(* CODESYS project TcDynStringKit.library
   Company: FisoThemes
   DefaultNamespace: TcDynStringKit
   Version: 1.0.1.1
   Placeholder: TwinCAT Dynamic String Kit
   Author: Goodwill Mzumala
   Description: A library that provides tools for working with dynamic strings in TwinCAT.
   Title: TwinCAT Dynamic String Kit

Project tree, tasks and I/O mapping:
  libraries: Tc2_Standard, * (Beckhoff Automation GmbH); Tc2_System, * (Beckhoff Automation GmbH); Tc2_Utilities, * (Beckhoff Automation GmbH); Tc3_Module, * (Beckhoff Automation GmbH)
  DUTs/
    Alias/
      data type T_Char
      data type T_LongString
      data type T_QueryInterface
      data type T_ShortString
      data type T_Size
      data type T_WhitespaceLocation
    Enums/
      data type E_WhitespaceLocation
    Structs/
    Unions/
  ITFs/
    Adapters/
      interface I_ReadOnlyLineBuilderAdapter
      interface I_ReadOnlyStringBuilderAdapter: Capacity, CopySubstringTo, CopyTo, GetBuffer, GetCapacity, GetChar, GetLength, GetString, GetSubstring, Length, Search, SearchAny, Split
      interface I_ReadOnlyWordBuilderAdapter
    Builders/
      interface I_LineBuilder
      interface I_StringBuilder: Append, AppendAny, AppendBuffer, AppendLine, BTrim, Capacity, Clear, CopySubstringTo, CopyTo, GetBuffer, GetCapacity, GetChar, GetLength, GetString, GetSubstring, Insert, InsertAny, InsertBuffer, Join, Length, LTrim, Remove, Replace, ReplaceAny, Reverse, RTrim, Search, SearchAny, Split, StrinkToFit, ToLowercase, ToUppercase
      interface I_WordBuilder
    Enumerators/
      interface I_Disposable: Dispose
      interface I_Enumerable: GetEnumerator
      interface I_Enumerator: Current, GetCurrent, Next, Reset
  PARAMs/
    GVLs/
      global variables Param_Configurations
  POUs/
    Examples/
      program P_AdapterExample [ST]
      program P_EnumeratorExample [ST]
      program P_StringBuilderExample [ST]
    Function Blocks/
      _Internal/
        function block FB_Free [ST]: FB_exit, FB_init
      Adapters/
        function block FB_ReadOnlyStringBuilderAdapter [ST]: Capacity, CopySubstringTo, CopyTo, GetBuffer, GetCapacity, GetChar, GetEnumerator, GetLength, GetString, GetSubstring, Length, Search, SearchAny, Split
      Builders/
        function block FB_StringBuilder [ST]: Free, Is_Space, Malloc, Reserve, Append, AppendAny, AppendBuffer, AppendLine, BTrim, Capacity, Clear, CopySubstringTo, CopyTo, GetBuffer, GetCapacity, GetChar, GetEnumerator, GetLength, GetString, GetSubstring, Insert, InsertAny, InsertBuffer, Join, Length, LTrim, Remove, Replace, ReplaceAny, Reverse, RTrim, Search, SearchAny, Split, StrinkToFit, ToLowercase, ToUppercase
      Enumerators/
        function block FB_AbstractStringEnumerator [ST]: Current, Dispose, GetCurrent, Next, Reset
        function block FB_StringBuilderEnumerator [ST]: Current, Current_Buffer, FB_init, GetCurrent, Next
    Functions/
      function F_AnyStringLength [ST]
      function F_AnyToString [ST]
      function F_ByteToChar [ST]
      function F_CharToByte [ST]
      function F_IsAnyToStringCompatable [ST]
      function F_IsBool [ST]
      function F_IsDigit [ST]
      function F_IsLTime [ST]
      function F_IsNumber [ST]
      function F_IsSignedInteger [ST]
      function F_IsSpace [ST]
      function F_IsTime [ST]
      function F_IsUnsignedInteger [ST]
      function F_MallocStr [ST]
      function F_MemCpy [ST]
      function F_MemMove [ST]
      function F_StringBuilder [ST]
      function F_StrLCat [ST]
      function F_StrLCpy [ST]
      function F_StrLen [ST]
      function F_StrNCmp [ST]
      function F_StrStr [ST]
      function F_StrToAny [ST]
      function F_ToLower [ST]
      function F_ToUpper [ST]
      function F_TrimWhiteSpace [ST]
    program MAIN [ST]
  Project Information/
    function F_GetCompany [ST]
    function F_GetTitle [ST]
    function F_GetVersion [ST]
  Version/
    global variables Global_Version
  VISUs/
*)

// DUTs/Alias/T_Char
TYPE T_Char : STRING(1); END_TYPE

// DUTs/Alias/T_LongString
TYPE T_LongString : STRING(Param_Configurations.LongStringSize); END_TYPE

// DUTs/Alias/T_QueryInterface
TYPE T_QueryInterface : __SYSTEM.IQueryInterface; END_TYPE

// DUTs/Alias/T_ShortString
TYPE T_ShortString : STRING(Param_Configurations.ShortStringSize); END_TYPE

// DUTs/Alias/T_Size
TYPE T_Size : DINT; END_TYPE

// DUTs/Alias/T_WhitespaceLocation
TYPE T_WhitespaceLocation : E_WhitespaceLocation; END_TYPE

// DUTs/Enums/E_WhitespaceLocation
{attribute 'qualified_only'}
{attribute 'to_string'}
TYPE E_WhitespaceLocation :
(
	Both := 0,
	Start,
	End
);
END_TYPE

// PARAMs/GVLs/Param_Configurations
{attribute 'qualified_only'}
VAR_GLOBAL CONSTANT
	ShortStringSize : UXINT := 80;
	LongStringSize : UXINT := 255;
END_VAR

// Version/Global_Version
{attribute 'TcGenerated'}
{attribute 'no-analysis'}
{attribute 'linkalways'}
// This function has been automatically generated from the project information.
VAR_GLOBAL CONSTANT
	{attribute 'const_non_replaced'}
	stLibVersion_TwinCAT_Dynamic_String_Kit : ST_LibVersion := (iMajor := 1, iMinor := 0, iBuild := 1, iRevision := 1, nFlags := 0, sVersion := '1.0.1.1');
END_VAR

// ITFs/Adapters/I_ReadOnlyLineBuilderAdapter
INTERFACE I_ReadOnlyLineBuilderAdapter EXTENDS T_QueryInterface

END_INTERFACE

// ITFs/Adapters/I_ReadOnlyStringBuilderAdapter
INTERFACE I_ReadOnlyStringBuilderAdapter EXTENDS T_QueryInterface

// Number of bytes allocated in memory for the string builder's contents.
PROPERTY Capacity : T_Size
GET
END_GET
END_PROPERTY

// Copies a subset of characters in the string builder from specified position at specified length to a string
METHOD CopySubstringTo : I_ReadOnlyStringBuilderAdapter
VAR_INPUT
	Position, Length : T_Size;
	Value : ANY;
END_VAR
END_METHOD

// Copies contents of string builder to given string of any size
METHOD CopyTo : I_ReadOnlyStringBuilderAdapter
VAR_INPUT
	Value : ANY;
END_VAR
END_METHOD

// !!!UNSAFE!!! DON'T FORGET TO RELEASE/DELETE FROM	MEMORY WHEN DONE!
// | Get a copy of the internal string buffer at the size of the string length + 1.
METHOD GetBuffer : I_ReadOnlyStringBuilderAdapter
VAR_IN_OUT
	pBuffer : POINTER TO BYTE;
END_VAR
END_METHOD

// Retrieves the number of bytes allocated in memory for the string builder's contents.
METHOD GetCapacity : I_ReadOnlyStringBuilderAdapter
VAR_OUTPUT
	Capacity : T_Size;
END_VAR
END_METHOD

// Gets character at specified position in the string builder
METHOD GetChar : T_Char
VAR_INPUT
	Position : T_Size;
END_VAR
END_METHOD

// Retrieves the current size of string builder contents
METHOD GetLength : I_ReadOnlyStringBuilderAdapter
VAR_OUTPUT
	Length : T_Size;
END_VAR
END_METHOD

// Converts contents of string builder to string and returns them
METHOD GetString : T_LongString
VAR_INPUT
END_VAR
END_METHOD

// Get a subset of characters in the string builder from specified position at specified length and returns them as a string
METHOD GetSubstring : T_LongString
VAR_INPUT
	Position, Length : T_Size;
END_VAR
END_METHOD

// Current size of string builder contents
PROPERTY Length : T_Size
GET
END_GET
END_PROPERTY

// Finds the position of the first instance of a given string in the content's of the string builder from a starting position
METHOD Search : I_ReadOnlyStringBuilderAdapter
VAR_INPUT
	sValue : T_LongString;
	Start_Position : T_Size;
END_VAR
VAR_OUTPUT
	Position : T_Size;
END_VAR
END_METHOD

// Finds the position of the first instance of a given value in the content's of the string builder from a starting position
METHOD SearchAny : I_ReadOnlyStringBuilderAdapter
VAR_INPUT
	Value : ANY;
	Start_Position : T_Size;
END_VAR
VAR_OUTPUT
	Position : T_Size := -1;
END_VAR
END_METHOD

// Appends selected characters from the current string builder to the selected string builder
METHOD Split : I_ReadOnlyStringBuilderAdapter
VAR_INPUT
	Position, Length : T_Size;
	ipStringBuilder : I_StringBuilder;
END_VAR
END_METHOD

END_INTERFACE

// ITFs/Builders/I_StringBuilder
INTERFACE I_StringBuilder EXTENDS T_QueryInterface

// Appends the given string to the end of the string builder's contents.
METHOD Append : I_StringBuilder
VAR_INPUT
	sValue : T_LongString;
END_VAR
END_METHOD

// Appends the given value to the end of the string builder's contents.
METHOD AppendAny : I_StringBuilder
VAR_INPUT
	Value : ANY;
END_VAR
END_METHOD

// !!!UNSAFE!!! THIS WILL APPEND UP TO THE NULL CHARACTER. IF NO NULL EXISTS, THIS WILL RUN FOREVER!
// | Append raw values directly to the internal string buffer. This is meant for appending dynamic strings to the string builder.
METHOD AppendBuffer : I_StringBuilder
VAR_INPUT
	pBuffer : POINTER TO BYTE;
END_VAR
END_METHOD

// Appends a new line (\r\n or $r$n) to string builder's contents.
METHOD AppendLine : I_StringBuilder
END_METHOD

// Removes all ASCII white space (spaces, tabs, carriage returns, and linefeeds) from the beginning and end of string in the string builder
METHOD BTrim : I_StringBuilder
END_METHOD

// Number of bytes allocated in memory for the string builder's contents.
PROPERTY Capacity : T_Size
GET
END_GET
END_PROPERTY

// Empties the string builder's contents, resetting its length to zero.
METHOD Clear : I_StringBuilder
END_METHOD

// Copies a subset of characters in the string builder from specified position at specified length to a string
METHOD CopySubstringTo : I_StringBuilder
VAR_INPUT
	Position, Length : T_Size;
	Value : ANY;
END_VAR
END_METHOD

// Copies contents of string builder to given string of any size
METHOD CopyTo : I_StringBuilder
VAR_INPUT
	Value : ANY;
END_VAR
END_METHOD

// !!!UNSAFE!!! DON'T FORGET TO RELEASE/DELETE FROM	MEMORY WHEN DONE!
// | Get a copy of the internal string buffer at the size of the string length + 1.
METHOD GetBuffer : I_StringBuilder
VAR_IN_OUT
	pBuffer : POINTER TO BYTE;
END_VAR
END_METHOD

// Retrieves the number of bytes allocated in memory for the string builder's contents.
METHOD GetCapacity : I_StringBuilder
VAR_OUTPUT
	Capacity : T_Size;
END_VAR
END_METHOD

// Gets character at specified position in the string builder
METHOD GetChar : T_Char
VAR_INPUT
	Position : T_Size;
END_VAR
END_METHOD

// Retrieves the current size of string builder contents
METHOD GetLength : I_StringBuilder
VAR_OUTPUT
	Length : T_Size;
END_VAR
END_METHOD

// Converts contents of string builder to string and returns them
METHOD GetString : T_LongString
VAR_INPUT
END_VAR
END_METHOD

// Get a subset of characters in the string builder from specified position at specified length and returns them as a string
METHOD GetSubstring : T_LongString
VAR_INPUT
	Position, Length : T_Size;
END_VAR
END_METHOD

// Inserts the given string at the specified position.
METHOD Insert : I_StringBuilder
VAR_INPUT
	Position : T_Size;
	sValue : T_LongString;
END_VAR
END_METHOD

// Inserts the given value at the specified position.
METHOD InsertAny : I_StringBuilder
VAR_INPUT
	Position : T_Size;
	Value : ANY;
END_VAR
END_METHOD

// !!!UNSAFE!!! THIS WILL INSERT UP TO THE NULL CHARACTER. IF NO NULL EXISTS, THIS WILL RUN FOREVER!
// | Inserts raw values directly to the internal string buffer at the specified position. This is meant for inserting dynamic strings to the string builder.
METHOD InsertBuffer : I_StringBuilder
VAR_INPUT
	Position : T_Size;
	pBuffer : POINTER TO BYTE;
END_VAR
END_METHOD

// Joins/Merges the string contents of the current string builder with that on the specified string builder at the specified position
METHOD Join : I_StringBuilder
VAR_INPUT
	Position : T_Size;
	ipString_Builder : I_StringBuilder;
END_VAR
END_METHOD

// Current size of string builder contents
PROPERTY Length : T_Size
GET
END_GET
END_PROPERTY

// Removes all ASCII white space (spaces, tabs, carriage returns, and linefeeds) from the beginning of string in the string builder
METHOD LTrim : I_StringBuilder
VAR_INPUT
END_VAR
END_METHOD

// Removes the characters in the string builder from specified position at specified length.
METHOD Remove : I_StringBuilder
VAR_INPUT
	Position, Length : T_Size;
END_VAR
END_METHOD

// Replaces the instance of the old string in the string builder with the new string.
// If bReplace_All = TRUE, all instances of the old string are placed, else only the first instance.
METHOD Replace : I_StringBuilder
VAR_INPUT
	sOld_Value,
	sNew_Value : T_LongString;
	bReplace_All : BOOL;
END_VAR
END_METHOD

// Replaces the instance of the old value in the string builder with the new value.
// If bReplace_All = TRUE, all instances of the old value are placed, else only the first instance.
METHOD ReplaceAny : I_StringBuilder
VAR_INPUT
	Old_Value : ANY;
	New_Value : ANY;
	bReplace_All : BOOL;
END_VAR
END_METHOD

// Reverses the string contents in the string builder
METHOD Reverse : I_StringBuilder
VAR_INPUT
END_VAR
END_METHOD

// Removes all ASCII white space (spaces, tabs, carriage returns, and linefeeds) from the end of string in the string builder
METHOD RTrim : I_StringBuilder
VAR_INPUT
END_VAR
END_METHOD

// Finds the position of the first instance of a given string in the content's of the string builder from a starting position
METHOD Search : I_StringBuilder
VAR_INPUT
	sValue : T_LongString;
	Start_Position : T_Size;
END_VAR
VAR_OUTPUT
	Position : T_Size;
END_VAR
END_METHOD

// Finds the position of the first instance of a given value in the content's of the string builder from a starting position
METHOD SearchAny : I_StringBuilder
VAR_INPUT
	Value : ANY;
	Start_Position : T_Size;
END_VAR
VAR_OUTPUT
	Position : T_Size := -1;
END_VAR
END_METHOD

// Appends selected characters from the current string builder to the selected string builder
METHOD Split : I_StringBuilder
VAR_INPUT
	Position, Length : T_Size;
	ipStringBuilder : I_StringBuilder;
END_VAR
END_METHOD

// Reduces the capacity of the string builder to match the size of its contents, potentially reducing memory usage.
METHOD StrinkToFit : I_StringBuilder
END_METHOD

// Converts all alphabetic characters in string builder to lowercase characters
METHOD ToLowercase : I_StringBuilder
VAR_INPUT
END_VAR
END_METHOD

// Converts all alphabetic characters in string builder to uppercase characters
METHOD ToUppercase : I_StringBuilder
VAR_INPUT
END_VAR
END_METHOD

END_INTERFACE

// ITFs/Adapters/I_ReadOnlyWordBuilderAdapter
INTERFACE I_ReadOnlyWordBuilderAdapter EXTENDS T_QueryInterface

END_INTERFACE

// ITFs/Builders/I_LineBuilder
INTERFACE I_LineBuilder EXTENDS T_QueryInterface

END_INTERFACE

// ITFs/Builders/I_WordBuilder
INTERFACE I_WordBuilder EXTENDS T_QueryInterface

END_INTERFACE

// ITFs/Enumerators/I_Disposable
INTERFACE I_Disposable EXTENDS T_QueryInterface

// Disposes or release resources for specified task
METHOD Dispose
VAR_INPUT
END_VAR
END_METHOD

END_INTERFACE

// ITFs/Enumerators/I_Enumerable
INTERFACE I_Enumerable EXTENDS T_QueryInterface

METHOD GetEnumerator : I_Enumerator
VAR_INPUT
END_VAR
END_METHOD

END_INTERFACE

// ITFs/Enumerators/I_Enumerator
INTERFACE I_Enumerator EXTENDS I_Disposable

(* Gets current string representation of element*)
PROPERTY Current : T_LongString
GET
END_GET
END_PROPERTY

// Gets current element. Returns TRUE if retrieval and converstion was successful.
METHOD GetCurrent : BOOL
VAR_INPUT
	sValue : REFERENCE TO STRING;
END_VAR
END_METHOD

// Advances enumerator to the next element. On first call or after reset it generates new element data to enumerate over.
METHOD Next : BOOL
VAR_INPUT
END_VAR
END_METHOD

// Sets enumerator to it's intial position. Disposes data pertaining to it's old elements.
METHOD Reset
VAR_INPUT
END_VAR
END_METHOD

END_INTERFACE

// POUs/Examples/P_AdapterExample
PROGRAM INTERNAL P_AdapterExample
VAR
	bStart				: BOOL;
	sValue 				: STRING(255);
	nPos				: T_Size;
	tTime 				: TIME :=  TIME();
	tTime2				: TIME;
	fbStringBuilder 	: FB_StringBuilder;
	fbReadOnlySB 		: FB_ReadOnlyStringBuilderAdapter;
	ipReadOnlySB 		: I_ReadOnlyStringBuilderAdapter;
END_VAR

fbReadOnlySB(ipStringBuilder := fbStringBuilder);
ipReadOnlySB := fbReadOnlySB;

IF bStart THEN
	bStart := FALSE;
	fbStringBuilder
		.Clear()
		.Append('   I love cats.')
		.Append('The time is: ').AppendAny(tTime).Append('.')
		.Append('   ')
		.BTrim();
	END_IF

sValue := ipReadOnlySB
			.Search('T#', 0, Position => nPos)
			.CopySubstringTo(nPos, tc2_Standard.LEN(TO_STRING(tTime)), tTime2)
			.GetString();

END_PROGRAM

// POUs/Function Blocks/Builders/FB_StringBuilder
{attribute 'no_assign'}
{attribute 'enable_dynamic_creation'}
{attribute 'no_explicit_call' := 'do not call this POU directly'}
FUNCTION_BLOCK FB_StringBuilder IMPLEMENTS I_StringBuilder, I_Enumerable
VAR CONSTANT
	Default_Capacity : T_Size := 256;
END_VAR
VAR
	{attribute 'hide'} 
	_Capacity : T_Size := THIS^.Default_Capacity;
	{attribute 'hide'} 
	_Length : T_Size := 0;
	_pBuffer : POINTER TO STRING := THIS^.Malloc(THIS^.Capacity);
END_VAR
VAR CONSTANT
	{attribute 'hide'} 
	_fbFree : FB_Free(THIS^._pBuffer) := ();
END_VAR

// Dealloocates String from memory
METHOD PROTECTED Free
VAR_INPUT
END_VAR
IF THIS^._pBuffer <> 0 THEN __DELETE(THIS^._pBuffer); END_IF
THIS^.Capacity := 0;
END_METHOD

METHOD PROTECTED Is_Space : BOOL
VAR_INPUT
	nChar : BYTE;
END_VAR
Is_Space := (nChar = 32) OR_ELSE (nChar = 9) OR_ELSE (nChar = 10) OR_ELSE (nChar = 13) OR_ELSE (nChar = 12) OR_ELSE (nChar = 11);
END_METHOD

// Allocates memory on the heap for a string of defined size
METHOD PROTECTED Malloc : POINTER TO STRING
VAR_INPUT
	Size : T_Size;
END_VAR
Malloc := __NEW(BYTE, TO_UDINT(Size));
END_METHOD

METHOD PROTECTED Reserve
VAR_INPUT
	Capacity : T_Size;
END_VAR
VAR
	pTemp : POINTER TO STRING;
END_VAR
IF Capacity <= THIS^.Capacity THEN RETURN; END_IF
pTemp := THIS^.Malloc(Capacity);
F_StrLCpy(pTemp, THIS^._pBuffer, Capacity);
THIS^.Free();
THIS^._pBuffer := pTemp;
THIS^.Capacity := Capacity;
END_METHOD

// Appends the given string to the end of the string builder's contents.
METHOD Append : I_StringBuilder
VAR_INPUT
	sValue : T_LongString;
END_VAR
Append := THIS^.AppendAny(sValue);
END_METHOD

// Appends the given value to the end of the string builder's contents.
METHOD AppendAny : I_StringBuilder
VAR_INPUT
	Value : ANY;
END_VAR
VAR
	bMalloced : BOOL := TRUE;
	Str_Len : T_Size;
	pValue : POINTER TO STRING;
END_VAR
AppendAny := THIS^;
CASE Value.TypeClass OF
	__SYSTEM.TYPE_CLASS.TYPE_STRING: 
		Str_Len := F_StrLen(Value.pValue);
		pValue := Value.pValue;
		bMalloced := FALSE;
		
	__SYSTEM.TYPE_CLASS.TYPE_WSTRING:
		Str_Len := TO_DINT(Tc2_Utilities.WLEN2(Value.pValue));
		pValue := THIS^.Malloc(Str_Len);
		Tc2_Utilities.WSTRING_TO_STRING2(pValue, Value.pValue, TO_UDINT(Str_Len));
		
	__SYSTEM.TYPE_CLASS.TYPE_BOOL,
	__SYSTEM.TYPE_CLASS.TYPE_BYTE,
	__SYSTEM.TYPE_CLASS.TYPE_WORD,
	__SYSTEM.TYPE_CLASS.TYPE_DWORD,
	__SYSTEM.TYPE_CLASS.TYPE_LWORD,
	__SYSTEM.TYPE_CLASS.TYPE_SINT,
	__SYSTEM.TYPE_CLASS.TYPE_INT,
	__SYSTEM.TYPE_CLASS.TYPE_DINT,
	__SYSTEM.TYPE_CLASS.TYPE_LINT,
	__SYSTEM.TYPE_CLASS.TYPE_USINT,
	__SYSTEM.TYPE_CLASS.TYPE_UINT,
	__SYSTEM.TYPE_CLASS.TYPE_UDINT,
	__SYSTEM.TYPE_CLASS.TYPE_ULINT,
	__SYSTEM.TYPE_CLASS.TYPE_REAL,
	__SYSTEM.TYPE_CLASS.TYPE_LREAL,
	__SYSTEM.TYPE_CLASS.TYPE_TIME,
	__SYSTEM.TYPE_CLASS.TYPE_LTIME,
	__SYSTEM.TYPE_CLASS.TYPE_DATE,
	__SYSTEM.TYPE_CLASS.TYPE_DATEANDTIME,
	__SYSTEM.TYPE_CLASS.TYPE_TIMEOFDAY,
	__SYSTEM.TYPE_CLASS.TYPE_POINTER:
		pValue := THIS^.Malloc(SIZEOF(T_LongString));
		pValue^ := F_AnyToString(Value);
		Str_Len := F_StrLen(pValue);
ELSE
	RETURN;
END_CASE

IF (THIS^.Length + Str_Len) >= THIS^.Capacity THEN
	THIS^.Reserve((THIS^.Length + Str_Len + 1)*2);
	END_IF

THIS^.Length := THIS^.Length + Str_Len;
F_StrLCat(THIS^._pBuffer, pValue, THIS^.Length + 1);

IF bMalloced THEN __DELETE(pValue); END_IF
END_METHOD

// !!!UNSAFE!!! THIS WILL APPEND UP TO THE NULL CHARACTER. IF NO NULL EXISTS, THIS WILL RUN FOREVER!
// | Append raw values directly to the internal string buffer. This is meant for appending dynamic strings to the string builder.
METHOD AppendBuffer : I_StringBuilder
VAR_INPUT
	pBuffer : POINTER TO BYTE;
END_VAR
VAR
	Str_Len : T_Size;
END_VAR
AppendBuffer := THIS^;
IF pBuffer = 0 THEN RETURN; END_IF
Str_Len := F_StrLen(pBuffer);

IF (THIS^.Length + Str_Len) >= THIS^.Capacity THEN
	THIS^.Reserve((THIS^.Length + Str_Len + 1)*2);
	END_IF
	
THIS^.Length := THIS^.Length + Str_Len;
F_StrLCat(THIS^._pBuffer, pBuffer, THIS^.Length + 1);
END_METHOD

// Appends a new line (\r\n or $r$n) to string builder's contents.
METHOD AppendLine : I_StringBuilder
AppendLine := THIS^;
THIS^.Append('$r$n');
END_METHOD

// Removes all ASCII white space (spaces, tabs, carriage returns, and linefeeds) from the beginning and end of string in the string builder
METHOD BTrim : I_StringBuilder
VAR
	Start, End, Length : T_Size := 0;
END_VAR
BTrim := THIS^;
IF THIS^.Length = 0 THEN RETURN; END_IF
End := THIS^.Length - 1;

WHILE ((Start <= End) AND THIS^.Is_Space(THIS^._pBuffer^[Start])) DO Start := Start  + 1; END_WHILE
WHILE ((End >= Start) AND THIS^.Is_Space(THIS^._pBuffer^[End])) DO End := End  - 1; END_WHILE

Length := end - start + 1;
F_MemMove(THIS^._pBuffer, ADR(THIS^._pBuffer^[Start]), Length);
THIS^.Length := Length;
THIS^._pBuffer^[THIS^.Length] := 0;
END_METHOD

// Number of bytes allocated in memory for the string builder's contents.
PROPERTY Capacity : T_Size
GET
Capacity := THIS^._Capacity;
END_GET
SET
PROTECTED
THIS^._Capacity := Capacity;
END_SET
END_PROPERTY

// Empties the string builder's contents, resetting its length to zero.
METHOD Clear : I_StringBuilder
Clear := THIS^;
THIS^.Free();
THIS^.Capacity := THIS^.Default_Capacity;
THIS^.Length := 0;
THIS^._pBuffer := THIS^.Malloc(THIS^.Capacity);
THIS^._pBuffer^[0] := 0;
END_METHOD

// Copies a subset of characters in the string builder from specified position at specified length to a string
METHOD CopySubstringTo : I_StringBuilder
VAR_INPUT
	Position, Length : T_Size;
	Value : ANY;
END_VAR
VAR
	pTemp : POINTER TO BYTE;
	pwsTemp : POINTER TO WSTRING;
END_VAR
CopySubstringTo := THIS^;
IF Value.pValue = 0 THEN RETURN; END_IF
CASE Value.TypeClass OF
	__SYSTEM.TYPE_CLASS.TYPE_STRING:
		Length := MIN(Length, Value.diSize - 1);
		IF (Position > THIS^.Length) OR_ELSE (Length <= 0) OR_ELSE (THIS^.Length = 0) THEN Value.pValue[0] := 0; RETURN; END_IF
		F_StrLCpy(Value.pValue, ADR(THIS^._pBuffer^[Position]), Length + 1);
		
	__SYSTEM.TYPE_CLASS.TYPE_WSTRING:
		Length := MIN(Length, (Value.diSize/2) - 1 );
		IF (Position > THIS^.Length) OR_ELSE (Length = 0) OR_ELSE (THIS^.Length = 0) THEN pwsTemp := Value.pValue; pwsTemp^ := ""; RETURN; END_IF
		pTemp := THIS^.Malloc(Length + 1);
		F_StrLCpy(pTemp, ADR(THIS^._pBuffer^[Position]), Length + 1);
		Tc2_Utilities.STRING_TO_WSTRING2(Value.pValue, pTemp, TO_UDINT((Length*2)+1));
		__DELETE(pTemp);
ELSE
	F_StrToAny(Value, THIS^.GetSubstring(Position, Length));
END_CASE
END_METHOD

// Copies contents of string builder to given string of any size
METHOD CopyTo : I_StringBuilder
VAR_INPUT
	Value : ANY;
END_VAR
CopyTo := THIS^;
IF THIS^._pBuffer = 0 THEN Value.pValue[0] := 0; RETURN; END_IF 
CASE Value.TypeClass OF
	__SYSTEM.TYPE_CLASS.TYPE_STRING:
		F_StrLCpy(Value.pValue, THIS^._pBuffer, Value.diSize);
	__SYSTEM.TYPE_CLASS.TYPE_WSTRING:
		Tc2_Utilities.STRING_TO_WSTRING2(Value.pValue, THIS^._pBuffer, TO_UDINT(Value.diSize));
ELSE
	F_StrToAny(Value, THIS^.GetString());
END_CASE
END_METHOD

// !!!UNSAFE!!! DON'T FORGET TO RELEASE/DELETE FROM	MEMORY WHEN DONE!
// | Get a copy of the internal string buffer at the size of the string length + 1.
METHOD GetBuffer : I_StringBuilder
VAR_IN_OUT
	pBuffer : POINTER TO BYTE;
END_VAR
GetBuffer := THIS^;
pBuffer := THIS^.Malloc(THIS^.Length + 1);
F_StrLCpy(pBuffer, THIS^._pBuffer, THIS^.Length + 1);
END_METHOD

// Retrieves the number of bytes allocated in memory for the string builder's contents.
METHOD GetCapacity : I_StringBuilder
VAR_OUTPUT
	Capacity : T_Size;
END_VAR
GetCapacity := THIS^;
Capacity := THIS^.Capacity;
END_METHOD

// Gets character at specified position in the string builder
METHOD GetChar : T_Char
VAR_INPUT
	Position : T_Size;
END_VAR
IF Position < 0 THEN RETURN; END_IF
IF Position > THIS^.Length THEN RETURN; END_IF
GetChar[0] := THIS^._pBuffer^[Position];
END_METHOD

METHOD GetEnumerator : I_Enumerator
VAR_INST
	fbEnumerator : FB_StringBuilderEnumerator(THIS^);
END_VAR
GetEnumerator := fbEnumerator;
END_METHOD

// Retrieves the current size of string builder contents
METHOD GetLength : I_StringBuilder
VAR_OUTPUT
	Length : T_Size;
END_VAR
GetLength := THIS^;
Length := THIS^.Length;
END_METHOD

// Converts contents of string builder to string and returns them
METHOD GetString : T_LongString
THIS^.CopyTo(GetString);
END_METHOD

// Get a subset of characters in the string builder from specified position at specified length and returns them as a string
METHOD GetSubstring : T_LongString
VAR_INPUT
	Position, Length : T_Size;
END_VAR
THIS^.CopySubstringTo(Position, Length, GetSubstring);
END_METHOD

// Inserts the given string at the specified position.
METHOD Insert : I_StringBuilder
VAR_INPUT
	Position : T_Size;
	sValue : T_LongString;
END_VAR
Insert := THIS^.InsertAny(Position, sValue);
END_METHOD

// Inserts the given value at the specified position.
METHOD InsertAny : I_StringBuilder
VAR_INPUT
	Position : T_Size;
	Value : ANY;
END_VAR
VAR
	bMalloced : BOOL := TRUE;
	Str_Len : T_Size;
	pValue : POINTER TO STRING;
END_VAR
InsertAny := THIS^;
IF Position < 0 OR Position > THIS^.Length THEN RETURN; END_IF 
CASE Value.TypeClass OF
	__SYSTEM.TYPE_CLASS.TYPE_STRING: 
		Str_Len := F_StrLen(Value.pValue);
		pValue := Value.pValue;
		bMalloced := FALSE;
	
	__SYSTEM.TYPE_CLASS.TYPE_WSTRING:
		Str_Len := TO_DINT(Tc2_Utilities.WLEN2(Value.pValue));
		pValue := THIS^.Malloc(Str_Len);
		Tc2_Utilities.WSTRING_TO_STRING2(pValue, Value.pValue, TO_UDINT(Str_Len));

	__SYSTEM.TYPE_CLASS.TYPE_BOOL,
	__SYSTEM.TYPE_CLASS.TYPE_BYTE,
	__SYSTEM.TYPE_CLASS.TYPE_WORD,
	__SYSTEM.TYPE_CLASS.TYPE_DWORD,
	__SYSTEM.TYPE_CLASS.TYPE_LWORD,
	__SYSTEM.TYPE_CLASS.TYPE_SINT,
	__SYSTEM.TYPE_CLASS.TYPE_INT,
	__SYSTEM.TYPE_CLASS.TYPE_DINT,
	__SYSTEM.TYPE_CLASS.TYPE_LINT,
	__SYSTEM.TYPE_CLASS.TYPE_USINT,
	__SYSTEM.TYPE_CLASS.TYPE_UINT,
	__SYSTEM.TYPE_CLASS.TYPE_UDINT,
	__SYSTEM.TYPE_CLASS.TYPE_ULINT,
	__SYSTEM.TYPE_CLASS.TYPE_REAL,
	__SYSTEM.TYPE_CLASS.TYPE_LREAL,
	__SYSTEM.TYPE_CLASS.TYPE_TIME,
	__SYSTEM.TYPE_CLASS.TYPE_LTIME,
	__SYSTEM.TYPE_CLASS.TYPE_DATE,
	__SYSTEM.TYPE_CLASS.TYPE_DATEANDTIME,
	__SYSTEM.TYPE_CLASS.TYPE_TIMEOFDAY,
	__SYSTEM.TYPE_CLASS.TYPE_POINTER:
		pValue := THIS^.Malloc(SIZEOF(T_LongString));
		pValue^ := F_AnyToString(Value);
		Str_Len := F_StrLen(pValue);
ELSE
	RETURN;
END_CASE

IF (THIS^.Length + Str_Len) >= THIS^.Capacity THEN
	THIS^.Reserve((THIS^.Length + Str_Len + 1)*2);
	END_IF

F_MemMove(THIS^._pBuffer + TO_UDINT(Position) + TO_UDINT(Str_Len), THIS^._pBuffer + TO_UDINT(Position), THIS^.Length - Position + 1);
F_MemCpy(THIS^._pBuffer + TO_UDINT(Position), pValue, Str_Len); 
THIS^.Length := THIS^.Length + Str_Len;

IF bMalloced THEN __DELETE(pValue); END_IF
END_METHOD

// !!!UNSAFE!!! THIS WILL INSERT UP TO THE NULL CHARACTER. IF NO NULL EXISTS, THIS WILL RUN FOREVER!
// | Inserts raw values directly to the internal string buffer at the specified position. This is meant for inserting dynamic strings to the string builder.
METHOD InsertBuffer : I_StringBuilder
VAR_INPUT
	Position : T_Size;
	pBuffer : POINTER TO BYTE;
END_VAR
VAR
	Str_Len : T_Size;
END_VAR
InsertBuffer := THIS^;
IF pBuffer = 0 OR Position < 0 OR Position > THIS^.Length THEN RETURN; END_IF
Str_Len := F_StrLen(pBuffer);

IF (THIS^.Length + Str_Len) >= THIS^.Capacity THEN
	THIS^.Reserve((THIS^.Length + Str_Len + 1)*2);
	END_IF

F_MemMove(THIS^._pBuffer + TO_UDINT(Position) + TO_UDINT(Str_Len), THIS^._pBuffer + TO_UDINT(Position), THIS^.Length - Position + 1);
F_MemCpy(THIS^._pBuffer + TO_UDINT(Position), pBuffer, Str_Len); 
THIS^.Length := THIS^.Length + Str_Len;
END_METHOD

// Joins/Merges the string contents of the current string builder with that on the specified string builder at the specified position
METHOD Join : I_StringBuilder
VAR_INPUT
	Position : T_Size;
	ipString_Builder : I_StringBuilder;
END_VAR
VAR
	pTemp : POINTER TO BYTE;
END_VAR
Join := THIS^;
IF ipString_Builder = 0 THEN RETURN; END_IF
ipString_Builder.GetBuffer(pTemp);
THIS^.InsertBuffer(Position, pTemp);
CASE Tc2_System.F_CheckMemoryArea(pTemp, 1) OF 
	E_TcMemoryArea.Dynamic: __DELETE(pTemp);
END_CASE
END_METHOD

// Current size of string builder contents
PROPERTY Length : T_Size
GET
VAR
	i : UDINT;
END_VAR
Length := THIS^._Length;
END_GET
SET
PROTECTED 
VAR
END_VAR
THIS^._Length := Length;
END_SET
END_PROPERTY

// Removes all ASCII white space (spaces, tabs, carriage returns, and linefeeds) from the beginning of string in the string builder
METHOD LTrim : I_StringBuilder
VAR
	Start, End, Length : T_Size := 0;
END_VAR
LTrim := THIS^;
IF THIS^.Length = 0 THEN RETURN; END_IF
End := THIS^.Length - 1;

WHILE ((Start <= End) AND THIS^.Is_Space(THIS^._pBuffer^[Start])) DO Start := Start + 1; END_WHILE

Length := end - start + 1;
F_MemMove(THIS^._pBuffer, ADR(THIS^._pBuffer^[Start]), Length);
THIS^.Length := Length;
THIS^._pBuffer^[THIS^.Length] := 0;
END_METHOD

// Removes the characters in the string builder from specified position at specified length.+
METHOD Remove : I_StringBuilder
VAR_INPUT
	Position, Length : T_Size;
END_VAR
Remove := THIS^;
IF Position + Length > THIS^.Length OR Position < 0 OR Length <= 0 OR Position > THIS^.Length THEN RETURN; END_IF
F_MemMove(ADR(THIS^._pBuffer^[Position]), ADR(THIS^._pBuffer^[Position + Length]), THIS^.Length - (Position + Length) + 1);
THIS^.Length := THIS^.Length - Length;
END_METHOD

// Replaces the instance of the old string in the string builder with the new string.
// If bReplace_All = TRUE, all instances of the old string are placed, else only the first instance.
METHOD Replace : I_StringBuilder
VAR_INPUT
	sOld_Value,
	sNew_Value : T_LongString;
	bReplace_All : BOOL;
END_VAR
Replace := THIS^.ReplaceAny(sOld_Value,sNew_Value, bReplace_All);
END_METHOD

// Replaces the instance of the old value in the string builder with the new value.
// If bReplace_All = TRUE, all instances of the old value are placed, else only the first instance.
METHOD ReplaceAny : I_StringBuilder
VAR_INPUT
	Old_Value : ANY;
	New_Value : ANY;
	bReplace_All : BOOL;
END_VAR
VAR
	Position, 
	Old_Str_Len,
	New_Str_len : T_Size;
END_VAR
ReplaceAny := THIS^;
IF NOT(F_IsAnyToStringCompatable(Old_Value)) OR_ELSE NOT(F_IsAnyToStringCompatable(New_Value)) THEN RETURN; END_IF

Old_Str_Len := F_AnyStringLength(Old_Value);
New_Str_Len := F_AnyStringLength(New_Value);

WHILE Position < THIS^.Length DO
	THIS^.SearchAny(Old_Value, Position, Position => Position);
	THIS^.Remove(Position, Old_Str_Len);
	THIS^.InsertAny(Position, New_Value);
	IF NOT bReplace_All OR Position < 0 THEN EXIT; END_IF
	Position := Position + New_Str_Len;
	END_WHILE
END_METHOD

// Reverses the string contents in the string builder
METHOD Reverse : I_StringBuilder
VAR
	i : T_Size;
	nTemp : BYTE;
END_VAR
Reverse := THIS^;
IF THIS^.Length <= 0 THEN RETURN; END_IF
FOR i := 0 TO (THIS^.Length/2)-1 DO
	nTemp := THIS^._pBuffer^[i];
	THIS^._pBuffer^[i] := THIS^._pBuffer^[THIS^.Length - i - 1];
	THIS^._pBuffer^[THIS^.Length - i - 1] := nTemp;
	END_FOR
END_METHOD

// Removes all ASCII white space (spaces, tabs, carriage returns, and linefeeds) from the end of string in the string builder
METHOD RTrim : I_StringBuilder
VAR
	Start, End, Length : T_Size := 0;
END_VAR
RTrim := THIS^;
IF THIS^.Length = 0 THEN RETURN; END_IF
End := THIS^.Length - 1;

WHILE ((End >= Start) AND THIS^.Is_Space(THIS^._pBuffer^[End])) DO End := End  - 1; END_WHILE

Length := end - start + 1;
F_MemMove(THIS^._pBuffer, ADR(THIS^._pBuffer^[Start]), Length);
THIS^.Length := Length;
THIS^._pBuffer^[THIS^.Length] := 0;
END_METHOD

// Finds the position of the first instance of a given string in the content's of the string builder from a starting position
METHOD Search : I_StringBuilder
VAR_INPUT
	sValue : T_LongString;
	Start_Position : T_Size;
END_VAR
VAR_OUTPUT
	Position : T_Size;
END_VAR
Search := THIS^.SearchAny(sValue,Start_Position, Position => Position);
END_METHOD

// Finds the position of the first instance of a given value in the content's of the string builder from a starting position
METHOD SearchAny : I_StringBuilder
VAR_INPUT
	Value : ANY;
	Start_Position : T_Size;
END_VAR
VAR_OUTPUT
	Position : T_Size := -1;
END_VAR
VAR
	bMalloced : BOOL := TRUE;
	Str_Len : T_Size;
	pValue, pLoc : POINTER TO STRING;
END_VAR
SearchAny := THIS^;
IF Start_Position < 0 OR Start_Position > THIS^.Length - 1 THEN RETURN; END_IF
CASE Value.TypeClass OF
	__SYSTEM.TYPE_CLASS.TYPE_STRING: 
		pValue := Value.pValue;
		bMalloced := FALSE;
		
	__SYSTEM.TYPE_CLASS.TYPE_WSTRING:
		Str_Len := TO_DINT(Tc2_Utilities.WLEN2(Value.pValue));
		pValue := THIS^.Malloc(Str_Len + 1);
		Tc2_Utilities.WSTRING_TO_STRING2(pValue, Value.pValue, TO_UDINT(Str_Len));
		
	__SYSTEM.TYPE_CLASS.TYPE_BOOL,
	__SYSTEM.TYPE_CLASS.TYPE_BYTE,
	__SYSTEM.TYPE_CLASS.TYPE_WORD,
	__SYSTEM.TYPE_CLASS.TYPE_DWORD,
	__SYSTEM.TYPE_CLASS.TYPE_LWORD,
	__SYSTEM.TYPE_CLASS.TYPE_SINT,
	__SYSTEM.TYPE_CLASS.TYPE_INT,
	__SYSTEM.TYPE_CLASS.TYPE_DINT,
	__SYSTEM.TYPE_CLASS.TYPE_LINT,
	__SYSTEM.TYPE_CLASS.TYPE_USINT,
	__SYSTEM.TYPE_CLASS.TYPE_UINT,
	__SYSTEM.TYPE_CLASS.TYPE_UDINT,
	__SYSTEM.TYPE_CLASS.TYPE_ULINT,
	__SYSTEM.TYPE_CLASS.TYPE_REAL,
	__SYSTEM.TYPE_CLASS.TYPE_LREAL,
	__SYSTEM.TYPE_CLASS.TYPE_TIME,
	__SYSTEM.TYPE_CLASS.TYPE_LTIME,
	__SYSTEM.TYPE_CLASS.TYPE_DATE,
	__SYSTEM.TYPE_CLASS.TYPE_DATEANDTIME,
	__SYSTEM.TYPE_CLASS.TYPE_TIMEOFDAY,
	__SYSTEM.TYPE_CLASS.TYPE_POINTER:
		pValue := THIS^.Malloc(SIZEOF(T_LongString));
		pValue^ := F_AnyToString(Value);
ELSE
	RETURN;
END_CASE
pLoc := F_StrStr(ADR(THIS^._pBuffer^[Start_Position]), pValue);
IF bMalloced THEN __DELETE(pValue); END_IF
IF pLoc = 0 THEN RETURN; END_IF
Position := TO_DINT(pLoc - THIS^._pBuffer);
END_METHOD

// Appends selected characters from the current string builder to the selected string builder
METHOD Split : I_StringBuilder
VAR_INPUT
	Position, Length : T_Size;
	ipStringBuilder : I_StringBuilder;
END_VAR
VAR
	Char : T_Char;
	i, End_Position : T_Size;
END_VAR
Split := THIS^;
IF ipStringBuilder = 0 THEN RETURN; END_IF
IF (Position > THIS^.Length) OR_ELSE (Length <= 0) OR_ELSE (THIS^.Length = 0) THEN RETURN; END_IF
End_Position := Position + Length;
IF End_Position > THIS^.Length THEN End_Position := THIS^.Length; END_IF

FOR i := Position TO End_Position - 1 DO
	Char[0] := THIS^._pBuffer^[i];
	ipStringBuilder.Append(Char);
	END_FOR
END_METHOD

// Reduces the capacity of the string builder to match the size of its contents, potentially reducing memory usage.
METHOD StrinkToFit : I_StringBuilder
VAR
	pTemp : POINTER TO STRING;
END_VAR
StrinkToFit := THIS^;
IF THIS^.Capacity > (THIS^.Length + 1) THEN
	pTemp := THIS^.Malloc(THIS^.Length + 1);
	F_StrLCpy(pTemp, THIS^._pBuffer, THIS^.Length + 1);
	THIS^.Free();
	THIS^._pBuffer := pTemp;
	THIS^.Capacity := THIS^.Length + 1;
	END_IF
END_METHOD

// Converts all alphabetic characters in string builder to lowercase characters
METHOD ToLowercase : I_StringBuilder
VAR
	i : T_Size;
END_VAR
ToLowercase := THIS^;
IF THIS^.Length = 0 THEN RETURN; END_IF
FOR i := 0 TO THIS^.Length - 1 DO 
	IF THIS^._pBuffer^[i] >= 65 AND THIS^._pBuffer^[i]<= 90 THEN 
		THIS^._pBuffer^[i] := THIS^._pBuffer^[i] + 32; 
		END_IF
	END_FOR
END_METHOD

// Converts all alphabetic characters in string builder to uppercase characters
METHOD ToUppercase : I_StringBuilder
VAR
	i : T_Size;
END_VAR
ToUppercase := THIS^;
IF THIS^.Length = 0 THEN RETURN; END_IF
FOR i := 0 TO THIS^.Length - 1 DO 
	IF THIS^._pBuffer^[i] >= 97 AND THIS^._pBuffer^[i]<= 122 THEN 
		THIS^._pBuffer^[i] := THIS^._pBuffer^[i] - 32; 
		END_IF
	END_FOR
END_METHOD

END_FUNCTION_BLOCK

// POUs/Function Blocks/_Internal/FB_Free
// Frees pointer when this instance of the FB leaves the scope;
{attribute 'no_explicit_call' := 'do not call this POU directly'}
FUNCTION_BLOCK INTERNAL FINAL FB_Free
VAR
	_pValue : REFERENCE TO POINTER TO BYTE;
END_VAR

METHOD FB_exit : BOOL
VAR_INPUT
	bInCopyCode : BOOL; // if TRUE, the exit method is called for exiting an instance that is copied afterwards (online change).
END_VAR
IF bInCopyCode THEN RETURN; END_IF
IF NOT __ISVALIDREF(THIS^._pValue) THEN RETURN; END_IF
IF THIS^._pValue <> 0 THEN __DELETE(THIS^._pValue); END_IF
END_METHOD

{attribute 'no_explicit_call' := 'do not call this POU directly'}
METHOD FB_init : BOOL
VAR_INPUT
	bInitRetains 	: BOOL; // if TRUE, the retain variables are initialized (warm start / cold start)
	bInCopyCode 	: BOOL;  // if TRUE, the instance afterwards gets moved into the copy code (online change)
	pValue 			: REFERENCE TO POINTER TO BYTE; // Pointer to be freed on exit
END_VAR
THIS^._pValue REF= pValue;
END_METHOD

END_FUNCTION_BLOCK

// POUs/Functions/F_StrLCpy
// Safe string copy. RETURNS string length of pSrc
// Never copies past Dst_Size or pSrc byte size which ever is smaller.
FUNCTION F_StrLCpy : T_Size
VAR_INPUT
	pDst : POINTER TO STRING; // Destination string
	pSrc : POINTER TO STRING; // Source string
	DstSize : T_Size; // Byte size of destnation string including the null character
END_VAR
VAR
	SrcLen, CopyLen : T_Size;
END_VAR

IF pDst = 0 OR pSrc = 0 THEN RETURN; END_IF
SrcLen := F_StrLen(pSrc);

IF DstSize <= 0 OR SrcLen <= 0 THEN F_StrLCpy := SrcLen; RETURN; END_IF

CopyLen := SEL(SrcLen < DstSize - 1, DstSize - 1,SrcLen); 

F_MemCpy(pDst, pSrc, CopyLen);
pDst^[CopyLen] := 0;
F_StrLCpy := SrcLen;

END_FUNCTION

// POUs/Functions/F_StrLen
// Gets the length of a string;
FUNCTION F_StrLen : T_Size
VAR_INPUT
	pString : POINTER TO STRING;
END_VAR
VAR
	i : T_Size := 0;
END_VAR

IF pString = 0 THEN RETURN; END_IF
WHILE pString^[i] <> 0 DO
	i := i + 1;
	END_WHILE
F_StrLen := i;

END_FUNCTION

// POUs/Functions/F_MemCpy
// Copies bytes from source to destnation at specified length.
FUNCTION F_MemCpy : POINTER TO BYTE
VAR_INPUT
	pDst,
	pSrc : POINTER TO BYTE;
	Size : T_Size; 
END_VAR
VAR
	i : T_Size := 0;
END_VAR

IF pDst = 0 OR pSrc = 0 OR Size <= 0 THEN RETURN; END_IF
FOR i := 0 TO Size - 1  DO pDst[i] := pSrc[i]; END_FOR
F_MemCpy := pDst;

END_FUNCTION

// POUs/Functions/F_AnyToString
// Converts any to string
FUNCTION F_AnyToString : T_LongString
VAR_INPUT
	 Value : ANY;
END_VAR
VAR	
	pBool			: POINTER TO BOOL;
    pByte			: POINTER TO BYTE;
    pWord			: POINTER TO WORD;
    pDWord			: POINTER TO DWORD;
    pLWord			: POINTER TO LWORD;
    pSint			: POINTER TO SINT;
    pInt			: POINTER TO INT;
    pDint			: POINTER TO DINT;
    pLint			: POINTER TO LINT;
    pUSint			: POINTER TO USINT;
    pUInt			: POINTER TO UINT;
    pUDint			: POINTER TO UDINT;
    pULint			: POINTER TO ULINT;
    pReal			: POINTER TO REAL;
    pLReal			: POINTER TO LREAL;
    pString			: POINTER TO T_LongString;
    pWString		: POINTER TO WSTRING;
    pTime			: POINTER TO TIME;
    pDate			: POINTER TO DATE;
    pDateAndTime	: POINTER TO DATE_AND_TIME;
    pTimeOfDay		: POINTER TO TIME_OF_DAY;
    pPointer		: PVOID;
	pLTime 			: POINTER TO LTIME;
END_VAR

IF Value.pValue = 0 THEN RETURN; END_IF;

CASE Value.TypeClass OF 
	__SYSTEM.TYPE_CLASS.TYPE_BOOL:
		pBool := Value.pValue;
		F_AnyToString := TO_STRING(pBool^);
		
    __SYSTEM.TYPE_CLASS.TYPE_BYTE:
		pByte := Value.pValue;
		F_AnyToString := TO_STRING(pByte^);
		
    __SYSTEM.TYPE_CLASS.TYPE_WORD:
		pWord := Value.pValue;
		F_AnyToString := TO_STRING(pWord^);
		
    __SYSTEM.TYPE_CLASS.TYPE_DWORD:
		pDWord := Value.pValue;
		F_AnyToString := TO_STRING(pDWord^);
		
    __SYSTEM.TYPE_CLASS.TYPE_LWORD:
		pLWord := Value.pValue;
		F_AnyToString := TO_STRING(pLWord^);
		
    __SYSTEM.TYPE_CLASS.TYPE_SINT:
		pSint := Value.pValue;
		F_AnyToString := TO_STRING(pSint^);
		
    __SYSTEM.TYPE_CLASS.TYPE_INT:
		pInt := Value.pValue;
		F_AnyToString := TO_STRING(pInt^);
		
    __SYSTEM.TYPE_CLASS.TYPE_DINT:
		pDint := Value.pValue;
		F_AnyToString := TO_STRING(pDint^);
		
    __SYSTEM.TYPE_CLASS.TYPE_LINT:
		pLint := Value.pValue;
		F_AnyToString := TO_STRING(pLint^);
		
    __SYSTEM.TYPE_CLASS.TYPE_USINT:
		pUSint := Value.pValue;
		F_AnyToString := TO_STRING(pUSint^);
		
    __SYSTEM.TYPE_CLASS.TYPE_UINT:
		pUInt := Value.pValue;
		F_AnyToString := TO_STRING(pUInt^);
		
    __SYSTEM.TYPE_CLASS.TYPE_UDINT:
		pUDint := Value.pValue;
		F_AnyToString := TO_STRING(pUDint^);
		
    __SYSTEM.TYPE_CLASS.TYPE_ULINT:
		pULint := Value.pValue;
		F_AnyToString := TO_STRING(pULint^);
		
   __SYSTEM.TYPE_CLASS.TYPE_REAL:
		pReal := Value.pValue;
		F_AnyToString := TO_STRING(pReal^);
		
    __SYSTEM.TYPE_CLASS.TYPE_LREAL:
		pLReal := Value.pValue;
		F_AnyToString := TO_STRING(pLReal^);
		
    __SYSTEM.TYPE_CLASS.TYPE_STRING:
		pString := Value.pValue;
		F_AnyToString := TO_STRING(pString^);
		
   __SYSTEM.TYPE_CLASS.TYPE_WSTRING:
		pWString := Value.pValue;
		F_AnyToString := TO_STRING(pWString^);
		
    __SYSTEM.TYPE_CLASS.TYPE_TIME:
		pTime := Value.pValue;
		F_AnyToString := TO_STRING(pTime^);
		
    __SYSTEM.TYPE_CLASS.TYPE_DATE:
		pDate := Value.pValue;
		F_AnyToString := TO_STRING(pDate^);
		
    __SYSTEM.TYPE_CLASS.TYPE_DATEANDTIME:
		pDateAndTime := Value.pValue;
		F_AnyToString := TO_STRING(pDateAndTime^);
		
    __SYSTEM.TYPE_CLASS.TYPE_TIMEOFDAY:
		pTimeOfDay := Value.pValue;
		F_AnyToString := TO_STRING(pTimeOfDay^);
	
	__SYSTEM.TYPE_CLASS.TYPE_POINTER:
		F_AnyToString := TO_STRING(Value.pValue);
		
	__SYSTEM.TYPE_CLASS.TYPE_LTIME:
		pLTime := Value.pValue;
		F_AnyToString := TO_STRING(pLTime^);
ELSE
	RETURN; 
END_CASE

END_FUNCTION

// POUs/Functions/F_StrLCat
// Safe string concat. RETURNS length of concatinated string.
// Concatinates up to destination size.
FUNCTION F_StrLCat : T_Size
VAR_INPUT
	pDst : POINTER TO STRING; // Destination string
	pSrc : POINTER TO STRING; // Source string     
	DstSize : T_Size; // Byte size of destnation string including the null character
END_VAR
VAR
	SrcLen, DstLen, CopyLen : T_Size;
END_VAR

IF pDst = 0 OR pSrc = 0 THEN RETURN; END_IF

DstLen := F_StrLen(pDst);
SrcLen := F_StrLen(pSrc);

IF DstSize <= 0 OR DstLen >= DstSize THEN F_StrLCat := SrcLen; RETURN; END_IF

CopyLen := DstSize - DstLen - 1;

F_MemCpy(pDst + TO_UDINT(DstLen), pSrc, CopyLen);
pDst^[DstLen + CopyLen] := 0;
F_StrLCat := DstLen + SrcLen;

END_FUNCTION

// POUs/Functions/F_MemMove
FUNCTION F_MemMove : POINTER TO BYTE
VAR_INPUT
	pDst,
	pSrc : POINTER TO BYTE;
	Size : T_Size; 
END_VAR
VAR
	i : T_Size := 0;
END_VAR

IF pDst = 0 OR pSrc = 0 OR Size <= 0 THEN RETURN; END_IF

IF pDst < pSrc THEN
	FOR i := 0 TO Size - 1  DO pDst[i] := pSrc[i]; END_FOR
ELSE
	FOR i := Size TO 1 BY -1 DO pDst[i-1] := pSrc[i-1]; END_FOR
	END_IF
F_MemMove := pDst;

END_FUNCTION

// POUs/Functions/F_StrToAny
// Converts string to any, returns TRUE if successful
FUNCTION F_StrToAny : BOOL
VAR_INPUT
	 Value : ANY;
	 sValue : T_LongString;
END_VAR
VAR	
	pBool			: POINTER TO BOOL;
    pByte			: POINTER TO BYTE;
    pWord			: POINTER TO WORD;
    pDWord			: POINTER TO DWORD;
    pLWord			: POINTER TO LWORD;
    pSint			: POINTER TO SINT;
    pInt			: POINTER TO INT;
    pDint			: POINTER TO DINT;
    pLint			: POINTER TO LINT;
    pUSint			: POINTER TO USINT;
    pUInt			: POINTER TO UINT;
    pUDint			: POINTER TO UDINT;
    pULint			: POINTER TO ULINT;
    pReal			: POINTER TO REAL;
    pLReal			: POINTER TO LREAL;
    pString			: POINTER TO T_LongString;
    pWString		: POINTER TO WSTRING;
    pTime			: POINTER TO TIME;
    pDate			: POINTER TO DATE;
    pDateAndTime	: POINTER TO DATE_AND_TIME;
    pTimeOfDay	: POINTER TO TIME_OF_DAY;
    pPointer		: POINTER TO PVOID;
	pLTime 			: POINTER TO LTIME;
END_VAR

F_StrToAny := TRUE;
IF Value.pValue = 0 THEN F_StrToAny := FALSE; RETURN; END_IF;

CASE Value.TypeClass OF 
	__SYSTEM.TYPE_CLASS.TYPE_BOOL:
		IF NOT F_IsBool(sValue) THEN F_StrToAny := FALSE; RETURN; END_IF
		pBool := Value.pValue;
		pBool^ := TO_BOOL(sValue);
		
    __SYSTEM.TYPE_CLASS.TYPE_BYTE:
		IF NOT F_IsUnsignedInteger(sValue) THEN F_StrToAny := FALSE; RETURN; END_IF
		pByte := Value.pValue;
		pByte^ := TO_BYTE(sValue);
		
    __SYSTEM.TYPE_CLASS.TYPE_WORD:
		IF NOT F_IsUnsignedInteger(sValue) THEN F_StrToAny := FALSE; RETURN; END_IF
		pWord := Value.pValue;
		pWord^ := TO_WORD(sValue);
		
    __SYSTEM.TYPE_CLASS.TYPE_DWORD:
		IF NOT F_IsUnsignedInteger(sValue) THEN F_StrToAny := FALSE; RETURN; END_IF
		pDWord := Value.pValue;
		pDWord^ := TO_DWORD(sValue);
		
    __SYSTEM.TYPE_CLASS.TYPE_LWORD:
		IF NOT F_IsUnsignedInteger(sValue) THEN F_StrToAny := FALSE; RETURN; END_IF
		pLWord := Value.pValue;
		pLWord^ := TO_LWORD(sValue);
		
    __SYSTEM.TYPE_CLASS.TYPE_SINT:
		IF NOT F_IsSignedInteger(sValue) THEN F_StrToAny := FALSE; RETURN; END_IF
		pSint := Value.pValue;
		pSint^ := TO_SINT(sValue);
		
    __SYSTEM.TYPE_CLASS.TYPE_INT:
		IF NOT F_IsSignedInteger(sValue) THEN F_StrToAny := FALSE; RETURN; END_IF
		pInt := Value.pValue;
		pInt^ := TO_INT(sValue);
		
    __SYSTEM.TYPE_CLASS.TYPE_DINT:
		IF NOT F_IsSignedInteger(sValue) THEN F_StrToAny := FALSE; RETURN; END_IF
		pDint := Value.pValue;
		pDint^ := TO_DINT(sValue);
		
    __SYSTEM.TYPE_CLASS.TYPE_LINT:
		IF NOT F_IsSignedInteger(sValue) THEN F_StrToAny := FALSE; RETURN; END_IF
		pLint := Value.pValue;
		pLint^ := TO_LINT(sValue);
		
    __SYSTEM.TYPE_CLASS.TYPE_USINT:
		IF NOT F_IsUnsignedInteger(sValue) THEN F_StrToAny := FALSE; RETURN; END_IF
		pUSint := Value.pValue;
		pUSint^ := TO_USINT(sValue);
		
    __SYSTEM.TYPE_CLASS.TYPE_UINT:
		IF NOT F_IsUnsignedInteger(sValue) THEN F_StrToAny := FALSE; RETURN; END_IF
		pUInt := Value.pValue;
		pUInt^ := TO_UINT(sValue);
		
    __SYSTEM.TYPE_CLASS.TYPE_UDINT:
		IF NOT F_IsUnsignedInteger(sValue) THEN F_StrToAny := FALSE; RETURN; END_IF
		pUDint := Value.pValue;
		pUDint^ := TO_UDINT(sValue);
		
    __SYSTEM.TYPE_CLASS.TYPE_ULINT:
		IF NOT F_IsUnsignedInteger(sValue) THEN F_StrToAny := FALSE; RETURN; END_IF
		pULint := Value.pValue;
		pULint^ := TO_ULINT(sValue);
		
   __SYSTEM.TYPE_CLASS.TYPE_REAL:
   		IF NOT F_IsNumber(sValue) THEN F_StrToAny := FALSE; RETURN; END_IF
		pReal := Value.pValue;
		pReal^ := TO_REAL(sValue);
		
    __SYSTEM.TYPE_CLASS.TYPE_LREAL:
		IF NOT F_IsNumber(sValue) THEN F_StrToAny := FALSE; RETURN; END_IF
		pLReal := Value.pValue;
		pLReal^ := TO_LREAL(sValue);
		
    __SYSTEM.TYPE_CLASS.TYPE_STRING:
		F_StrLCpy(Value.pValue, ADR(sValue),Value.diSize); 
		
   __SYSTEM.TYPE_CLASS.TYPE_WSTRING:
   		Tc2_Utilities.STRING_TO_WSTRING2(Value.pValue, ADR(sValue), TO_UDINT(Value.diSize));
		
    __SYSTEM.TYPE_CLASS.TYPE_TIME:
		IF NOT F_IsTime(sValue) THEN RETURN; END_IF
		pTime := Value.pValue;
		pTime^ := TO_TIME(sValue);
		
	__SYSTEM.TYPE_CLASS.TYPE_LTIME:
		IF NOT F_IsLTime(sValue) THEN RETURN; END_IF
		pLTime := Value.pValue;
		pLTime^ := TO_LTIME(sValue);
		
    __SYSTEM.TYPE_CLASS.TYPE_DATE:
		pDate := Value.pValue;
		pDate^ := TO_DATE(sValue);
		
    __SYSTEM.TYPE_CLASS.TYPE_DATEANDTIME:
		pDateAndTime := Value.pValue;
		pDateAndTime^ := TO_DT(sValue);
		
    __SYSTEM.TYPE_CLASS.TYPE_TIMEOFDAY:
		pTimeOfDay := Value.pValue;
		pTimeOfDay^ := TO_TOD(sValue);
	
	__SYSTEM.TYPE_CLASS.TYPE_POINTER:
		pPointer := Value.pValue;
		pPointer^ := Tc2_Utilities.STRING_TO_PVOID(sValue);
		
ELSE
	F_StrToAny := FALSE;
END_CASE

END_FUNCTION

// POUs/Functions/F_IsBool
// Checks if string is boolean
FUNCTION F_IsBool : BOOL
VAR_INPUT
	sValue : T_LongString;
END_VAR
VAR
END_VAR

F_ToUpper(sValue);
F_IsBool := sValue = 'FALSE' OR_ELSE sValue = 'TRUE';

END_FUNCTION

// POUs/Functions/F_ToUpper
// Converts all alphabetic characters in a string uppercase characters
FUNCTION F_ToUpper
VAR_INPUT
	sValue : REFERENCE TO STRING; // String of any size
END_VAR
VAR
	i : T_Size;
END_VAR

WHILE sValue[i] <> 0 DO 
	IF sValue[i] >= 97 AND sValue[i]<= 122 THEN sValue[i] := sValue[i] - 32; END_IF
	i := i + 1;
	END_WHILE

END_FUNCTION

// POUs/Functions/F_IsUnsignedInteger
// Checks if a string is an unsigned interger
FUNCTION F_IsUnsignedInteger : BOOL
VAR_INPUT
	sValue : REFERENCE TO STRING;
END_VAR
VAR
	i : T_Size;
END_VAR

IF NOT F_IsDigit(F_ByteToChar(sValue[0])) THEN RETURN; END_IF
WHILE F_IsSpace(F_ByteToChar(sValue[i])) DO i := i + 1; END_WHILE
WHILE F_IsDigit(F_ByteToChar(sValue[i])) DO i := i + 1; END_WHILE
F_IsUnsignedInteger := sValue[i] = 0;

END_FUNCTION

// POUs/Functions/F_IsDigit
// Checks if a character is a digit
FUNCTION F_IsDigit : BOOL
VAR_INPUT
	Char : T_Char;
END_VAR

F_IsDigit := Char >= '0' AND Char <= '9';

END_FUNCTION

// POUs/Functions/F_ByteToChar
// Converts a BYTE to an ascii character
FUNCTION F_ByteToChar : T_Char
VAR_INPUT
	nByte : BYTE;
END_VAR

F_ByteToChar[0] := nByte;

END_FUNCTION

// POUs/Functions/F_IsSpace
// Checks if a character is ' '(space) '$t' (horizontal tab) '$n' (newline) '$r' (carriage return) '$f' (form feed) '$v' (vertical tab)
FUNCTION F_IsSpace : BOOL
VAR_INPUT
	Char : T_Char;
END_VAR

F_IsSpace := (Char[0] = 32) OR_ELSE (Char[0] = 9) OR_ELSE (Char[0] = 10) OR_ELSE (Char[0] = 13) OR_ELSE (Char[0] = 12) OR_ELSE (Char[0] = 11);

END_FUNCTION

// POUs/Functions/F_IsSignedInteger
// Checks if a string is a signed integer
FUNCTION F_IsSignedInteger : BOOL
VAR_INPUT
	sValue : REFERENCE TO STRING;
END_VAR
VAR
	i : T_Size;
END_VAR

IF F_ByteToChar(sValue[0]) = '+' OR_ELSE F_ByteToChar(sValue[0]) = '-' THEN i := i + 1; END_IF
IF NOT F_IsDigit(F_ByteToChar(sValue[i])) THEN RETURN; END_IF
WHILE F_IsSpace(F_ByteToChar(sValue[i])) DO i := i + 1; END_WHILE
WHILE F_IsDigit(F_ByteToChar(sValue[i])) DO i := i + 1; END_WHILE
F_IsSignedInteger := sValue[i] = 0;

END_FUNCTION

// POUs/Functions/F_IsNumber
// Checks is a string is a number
FUNCTION F_IsNumber : BOOL
VAR_INPUT
	sValue : REFERENCE TO STRING;
END_VAR
VAR
	i : T_Size;
	bHasDigits, bHasDecimal, bHasExponent : BOOL;
END_VAR

IF F_ByteToChar(sValue[0]) = '+' OR_ELSE F_ByteToChar(sValue[0]) = '-' THEN i := i + 1; END_IF
IF NOT F_IsDigit(F_ByteToChar(sValue[0])) THEN RETURN; END_IF
WHILE F_IsSpace(F_ByteToChar(sValue[i])) DO i := i + 1; END_WHILE
WHILE sValue[i] <> 0 DO
	IF F_IsDigit(F_ByteToChar(sValue[i])) THEN 
		bHasDigits := TRUE;
	ELSIF F_ByteToChar(sValue[i]) = '.' THEN
		IF bHasDecimal THEN RETURN; END_IF
		bHasDecimal := TRUE;
	ELSIF F_ByteToChar(sValue[i]) = 'E' OR_ELSE F_ByteToChar(sValue[i]) = 'e' THEN
		IF bHasExponent THEN RETURN; END_IF
		IF F_ByteToChar(sValue[i+1]) = '+' OR_ELSE F_ByteToChar(sValue[i+1]) = '-' THEN i := i + 1; END_IF
		bHasExponent := TRUE;
	ELSE
		RETURN; 
		END_IF
	i := i + 1; 
	END_WHILE

IF NOT bHasDigits THEN RETURN; END_IF
F_IsNumber := TRUE;

END_FUNCTION

// POUs/Functions/F_IsTime
// Checks if string is in the format of the IEC-61131 time datatype format
FUNCTION F_IsTime : BOOL
VAR_INPUT
	sValue : REFERENCE TO STRING;
END_VAR
VAR
	i, Length : T_Size;
	pTemp : POINTER TO STRING;
	sT_Sharp : STRING := 'T#';
	sTime_Sharp : STRING := 'TIME#';
	bHas_D,
	bHas_H,
	bHas_M,
	bHas_S,
	bHas_MS : BOOL;
END_VAR

Length := F_StrLen(ADR(sValue));
pTemp := F_MallocStr(Length+1);
F_StrLCpy(pTemp, ADR(sValue), Length+1);
F_ToUpper(pTemp^);

IF NOT(F_StrNCmp(pTemp^, sT_Sharp, 2)) AND_THEN NOT(F_StrNCmp(pTemp^, sTime_Sharp, 5)) THEN __DELETE(pTemp); RETURN; END_IF
__DELETE(pTemp);


FOR i := SEL(F_ByteToChar(sValue[1]) = '#', 5, 2) TO Length - 1 DO
	CASE sValue[i] OF
		68,100: // Check for D/d
			IF NOT F_IsDigit(F_ByteToChar(sValue[i-1])) THEN RETURN; END_IF
			IF bHas_D OR_ELSE bHas_H OR_ELSE bHas_M OR_ELSE bHas_S OR_ELSE bHas_MS THEN RETURN; END_IF
			bHas_D := TRUE;
		72,104: // Check for H/h
			IF NOT F_IsDigit(F_ByteToChar(sValue[i-1])) THEN RETURN; END_IF
			IF bHas_H OR_ELSE bHas_M OR_ELSE bHas_S OR_ELSE bHas_MS THEN RETURN; END_IF
			bHas_H := TRUE;
		77,109: // Check for M/m
			IF NOT F_IsDigit(F_ByteToChar(sValue[i-1])) THEN RETURN; END_IF
			IF sValue[i+1] = 83 OR_ELSE sValue[i+1] = 115 THEN
				IF bHas_MS THEN RETURN; END_IF;
				bHas_MS := TRUE;
			ELSE
				IF bHas_M OR_ELSE bHas_S OR_ELSE bHas_MS THEN RETURN; END_IF
				bHas_M := TRUE;
				END_IF
		83,115: // Check for S/s
			IF sValue[i-1] = 77 OR_ELSE sValue[i-1] = 109 THEN CONTINUE; END_IF
			IF NOT F_IsDigit(F_ByteToChar(sValue[i-1])) THEN RETURN; END_IF
			IF bHas_S OR_ELSE bHas_MS THEN RETURN; END_IF
			bHas_S := TRUE;
	ELSE
		IF F_IsDigit(F_ByteToChar(sValue[i])) THEN CONTINUE; END_IF
		RETURN;
	END_CASE
END_FOR

IF F_IsDigit(F_ByteToChar(sValue[i-1])) THEN RETURN; END_IF
F_IsTime := TRUE;

END_FUNCTION

// POUs/Functions/F_MallocStr
// Allocates memory on the heap for a string of defined size.
FUNCTION F_MallocStr : POINTER TO STRING
VAR_INPUT
	Size : T_Size; // Size in bytes
END_VAR

F_MallocStr := __NEW(BYTE, TO_UDINT(Size));

END_FUNCTION

// POUs/Functions/F_StrNCmp
// Compares n number of characters in a string to determine if theyre the same and returns true if they are.
FUNCTION F_StrNCmp : BOOL
VAR_INPUT
	sValue1, sValue2 : REFERENCE TO STRING; // String of any size
	Size : T_Size; // Number of characters to compare
END_VAR
VAR
	i : T_Size;
END_VAR

IF Size < 1 THEN RETURN; END_IF
FOR i := 0 TO Size - 1 DO
	IF (sValue1[i] = 0 AND sValue2[i] = 0) THEN EXIT; END_IF
	IF (sValue1[i] <> sValue2[i]) OR_ELSE (sValue1[i] = 0 OR sValue2[i] = 0) THEN RETURN; END_IF
	END_FOR
F_StrNCmp := TRUE;

END_FUNCTION

// POUs/Functions/F_IsLTime
// Checks if string is in the format of the IEC-61131 ltime datatype format
FUNCTION F_IsLTime : BOOL
VAR_INPUT
	sValue : REFERENCE TO STRING;
END_VAR
VAR
	i, Length : T_Size;
	pTemp : POINTER TO STRING;
	sLTime_Sharp : STRING := 'LTIME#';
	bHas_D,
	bHas_H,
	bHas_M,
	bHas_S,
	bHas_MS,
	bHas_NS : BOOL;
END_VAR

Length := F_StrLen(ADR(sValue));
pTemp := F_MallocStr(Length+1);
F_StrLCpy(pTemp, ADR(sValue), Length+1);
F_ToUpper(pTemp^);
IF NOT(F_StrNCmp(pTemp^, sLTime_Sharp, 6)) THEN __DELETE(pTemp); RETURN; END_IF
__DELETE(pTemp);

FOR i := 6 TO Length-1 DO
	CASE sValue[i] OF
		68,100: // Check for D/d
			IF NOT F_IsDigit(F_ByteToChar(sValue[i-1])) THEN RETURN; END_IF
			IF bHas_D OR_ELSE bHas_H OR_ELSE bHas_M OR_ELSE bHas_S OR_ELSE bHas_MS OR_ELSE bHas_NS THEN RETURN; END_IF
			bHas_D := TRUE;
		72,104: // Check for H/h
			IF NOT F_IsDigit(F_ByteToChar(sValue[i-1])) THEN RETURN; END_IF
			IF bHas_H OR_ELSE bHas_M OR_ELSE bHas_S OR_ELSE bHas_MS OR_ELSE bHas_NS THEN RETURN; END_IF
			bHas_H := TRUE;
		77,109: // Check for M/m
			IF NOT F_IsDigit(F_ByteToChar(sValue[i-1])) THEN RETURN; END_IF
			IF sValue[i+1] = 83 OR_ELSE sValue[i+1] = 115 THEN
				IF bHas_MS OR_ELSE bHas_NS THEN RETURN; END_IF;
				bHas_MS := TRUE;
			ELSE
				IF bHas_M OR_ELSE bHas_S OR_ELSE bHas_MS OR_ELSE bHas_NS THEN RETURN; END_IF
				bHas_M := TRUE;
				END_IF
		83,115: // Check for S/s
			IF sValue[i-1] = 77 OR_ELSE sValue[i-1] = 109 THEN CONTINUE; END_IF
			IF sValue[i-1] = 78 OR_ELSE sValue[i-1] = 110 THEN CONTINUE; END_IF
			IF NOT F_IsDigit(F_ByteToChar(sValue[i-1])) THEN RETURN; END_IF
			IF bHas_S OR_ELSE bHas_MS OR_ELSE bHas_NS THEN RETURN; END_IF
			bHas_S := TRUE;
		78, 110: // Check for N/n
			IF NOT F_IsDigit(F_ByteToChar(sValue[i-1])) THEN RETURN; END_IF
			IF bHas_NS THEN RETURN; END_IF
			IF sValue[i+1] = 83 OR_ELSE sValue[i+1] = 115 THEN bHas_NS := TRUE; CONTINUE; END_IF
			RETURN;
	ELSE
		IF F_IsDigit(F_ByteToChar(sValue[i])) THEN CONTINUE; END_IF
		RETURN;
	END_CASE
END_FOR
IF F_IsDigit(F_ByteToChar(sValue[i-1])) THEN RETURN; END_IF
F_IsLTime := TRUE;

END_FUNCTION

// POUs/Function Blocks/Enumerators/FB_StringBuilderEnumerator
FUNCTION_BLOCK FB_StringBuilderEnumerator EXTENDS FB_AbstractStringEnumerator
VAR
	_ipStringBuilder : I_StringBuilder; 
END_VAR

(* Gets current string element*)
PROPERTY Current : T_LongString
GET
IF THIS^._ipStringBuilder = 0 THEN RETURN; END_IF
Current := THIS^._ipStringBuilder.GetChar(THIS^._Index);
END_GET
END_PROPERTY

(* !!!UNSAFE!!! DON'T FORGET TO RELEASE/DELETE FROM	MEMORY WHEN DONE!
 | Get a copy of the current element as a string buffer whose size is string length + 1.*)
METHOD Current_Buffer
VAR_IN_OUT
	pBuffer	: POINTER TO BYTE;
END_VAR
VAR
	pTemp : POINTER TO STRING;
END_VAR
IF THIS^._ipStringBuilder = 0 OR THIS^._Index < 0 OR_ELSE THIS^._Index >= THIS^._ipStringBuilder.Length THEN RETURN; END_IF
pTemp := __NEW(BYTE, 2);
pTemp^ := THIS^._ipStringBuilder.GetChar(THIS^._Index);
END_METHOD

{attribute 'hide'}
METHOD FB_init : BOOL
VAR_INPUT
	bInitRetains : BOOL; // if TRUE, the retain variables are initialized (warm start / cold start)
	bInCopyCode : BOOL;  // if TRUE, the instance afterwards gets moved into the copy code (online change)
	ipStringBuilder : I_StringBuilder;
END_VAR
THIS^._ipStringBuilder := ipStringBuilder;
END_METHOD

(* Gets current element. Returns TRUE if retrieval and converstion was successful. *)
METHOD GetCurrent : BOOL
VAR_INPUT
	sValue : REFERENCE TO STRING;
END_VAR
IF THIS^._ipStringBuilder = 0 THEN RETURN; END_IF
sValue := THIS^._ipStringBuilder.GetChar(THIS^._Index);
GetCurrent := TRUE;
END_METHOD

(* Advances enumerator to the next element. On first call or after reset it generates new element data to enumerate over.*)
METHOD Next : BOOL
IF THIS^._ipStringBuilder = 0 OR_ELSE THIS^._Index >= THIS^._ipStringBuilder.Length THEN RETURN; END_IF
THIS^._Index := THIS^._Index + 1;
Next := TRUE;
END_METHOD

END_FUNCTION_BLOCK

// POUs/Function Blocks/Enumerators/FB_AbstractStringEnumerator
FUNCTION_BLOCK ABSTRACT FB_AbstractStringEnumerator IMPLEMENTS I_Enumerator
VAR
	_Index : T_Size := -1;
END_VAR

(* Gets current string representation of element*)
PROPERTY ABSTRACT Current : T_LongString
GET
END_GET
END_PROPERTY

(* Disposes or release resources for specified task*)
METHOD Dispose
END_METHOD

(* Gets current element. Returns TRUE if retrieval and converstion was successful.*)
METHOD ABSTRACT GetCurrent : BOOL
VAR_INPUT
	sValue : REFERENCE TO STRING;
END_VAR
END_METHOD

(* Advances enumerator to the next element. On first call or after reset it generates new element data to enumerate over.*)
METHOD ABSTRACT Next : BOOL
END_METHOD

(* Sets enumerator to it's intial position. Disposes data pertaining to it's old elements.*)
METHOD Reset
THIS^._Index := -1;
END_METHOD

END_FUNCTION_BLOCK

// POUs/Functions/F_IsAnyToStringCompatable
// Checks if value can be converted to string
FUNCTION F_IsAnyToStringCompatable : BOOL
VAR_INPUT
	Value : ANY;
END_VAR

CASE Value.TypeClass OF
	__SYSTEM.TYPE_CLASS.TYPE_STRING,
	__SYSTEM.TYPE_CLASS.TYPE_WSTRING,
	__SYSTEM.TYPE_CLASS.TYPE_BOOL,
	__SYSTEM.TYPE_CLASS.TYPE_BYTE,
	__SYSTEM.TYPE_CLASS.TYPE_WORD,
	__SYSTEM.TYPE_CLASS.TYPE_DWORD,
	__SYSTEM.TYPE_CLASS.TYPE_LWORD,
	__SYSTEM.TYPE_CLASS.TYPE_SINT,
	__SYSTEM.TYPE_CLASS.TYPE_INT,
	__SYSTEM.TYPE_CLASS.TYPE_DINT,
	__SYSTEM.TYPE_CLASS.TYPE_LINT,
	__SYSTEM.TYPE_CLASS.TYPE_USINT,
	__SYSTEM.TYPE_CLASS.TYPE_UINT,
	__SYSTEM.TYPE_CLASS.TYPE_UDINT,
	__SYSTEM.TYPE_CLASS.TYPE_ULINT,
	__SYSTEM.TYPE_CLASS.TYPE_REAL,
	__SYSTEM.TYPE_CLASS.TYPE_LREAL,
	__SYSTEM.TYPE_CLASS.TYPE_TIME,
	__SYSTEM.TYPE_CLASS.TYPE_LTIME,
	__SYSTEM.TYPE_CLASS.TYPE_DATE,
	__SYSTEM.TYPE_CLASS.TYPE_DATEANDTIME,
	__SYSTEM.TYPE_CLASS.TYPE_TIMEOFDAY,
	__SYSTEM.TYPE_CLASS.TYPE_POINTER:
		F_IsAnyToStringCompatable := TRUE;
ELSE
	RETURN;
END_CASE

END_FUNCTION

// POUs/Functions/F_AnyStringLength
// Get the length of any value if converted to string
FUNCTION F_AnyStringLength : T_Size
VAR_INPUT
	Value : ANY;
END_VAR
VAR
	nSz : UDINT;
	pTemp : POINTER TO STRING;
END_VAR

CASE Value.TypeClass OF
	__SYSTEM.TYPE_CLASS.TYPE_STRING: 
		F_AnyStringLength := F_StrLen(Value.pValue);
		
	__SYSTEM.TYPE_CLASS.TYPE_WSTRING:
		F_AnyStringLength := TO_DINT(Tc2_Utilities.WLEN2(Value.pValue));
		
	__SYSTEM.TYPE_CLASS.TYPE_BOOL,
	__SYSTEM.TYPE_CLASS.TYPE_BYTE,
	__SYSTEM.TYPE_CLASS.TYPE_WORD,
	__SYSTEM.TYPE_CLASS.TYPE_DWORD,
	__SYSTEM.TYPE_CLASS.TYPE_LWORD,
	__SYSTEM.TYPE_CLASS.TYPE_SINT,
	__SYSTEM.TYPE_CLASS.TYPE_INT,
	__SYSTEM.TYPE_CLASS.TYPE_DINT,
	__SYSTEM.TYPE_CLASS.TYPE_LINT,
	__SYSTEM.TYPE_CLASS.TYPE_USINT,
	__SYSTEM.TYPE_CLASS.TYPE_UINT,
	__SYSTEM.TYPE_CLASS.TYPE_UDINT,
	__SYSTEM.TYPE_CLASS.TYPE_ULINT,
	__SYSTEM.TYPE_CLASS.TYPE_REAL,
	__SYSTEM.TYPE_CLASS.TYPE_LREAL,
	__SYSTEM.TYPE_CLASS.TYPE_TIME,
	__SYSTEM.TYPE_CLASS.TYPE_LTIME,
	__SYSTEM.TYPE_CLASS.TYPE_DATE,
	__SYSTEM.TYPE_CLASS.TYPE_DATEANDTIME,
	__SYSTEM.TYPE_CLASS.TYPE_TIMEOFDAY,
	__SYSTEM.TYPE_CLASS.TYPE_POINTER:
		F_AnyStringLength := Tc2_Standard.LEN(F_AnyToString(Value));
ELSE
	RETURN;
END_CASE

END_FUNCTION

// POUs/Functions/F_StrStr
// Searches for the first occurrence of a substring within a string. (Needle in a haystack)
// If found, a pointer to the first character of the substring within the original string is returned, else a null pointer is returned.
FUNCTION F_StrStr : POINTER TO STRING
VAR_INPUT
	pHaystackStr,
	pNeedleStr : POINTER TO STRING; 
END_VAR
VAR
	i,j, HaystackLen, NeedleLen : T_Size;
END_VAR

IF pHaystackStr = 0 OR pNeedleStr = 0 THEN RETURN; END_IF

HaystackLen := F_StrLen(pHaystackStr);
NeedleLen := F_StrLen(pNeedleStr);

IF NeedleLen > HaystackLen THEN RETURN; END_IF

FOR i := 0 TO HaystackLen - NeedleLen DO 
	FOR j := 0 TO NeedleLen - 1 DO 
		IF pHaystackStr^[i+j] <> pNeedleStr^[j] THEN EXIT; END_IF
		END_FOR
	IF j = NeedleLen THEN F_StrStr := pHaystackStr + TO_UDINT(i); RETURN; END_IF
	END_FOR

END_FUNCTION

// POUs/Function Blocks/Adapters/FB_ReadOnlyStringBuilderAdapter
FUNCTION_BLOCK FB_ReadOnlyStringBuilderAdapter IMPLEMENTS I_ReadOnlyStringBuilderAdapter, I_Enumerable
VAR_INPUT
	ipStringBuilder : I_StringBuilder;
END_VAR

(* Number of bytes allocated in memory for the string builder's contents.*)
PROPERTY Capacity : T_Size
GET
IF THIS^.ipStringBuilder = 0 THEN RETURN; END_IF
Capacity := THIS^.ipStringBuilder.Capacity;
END_GET
END_PROPERTY

(* Copies a subset of characters in the string builder from specified position at specified length to a string*)
METHOD CopySubstringTo : I_ReadOnlyStringBuilderAdapter
VAR_INPUT
	Position, Length : T_Size;
	Value : ANY;
END_VAR
CopySubstringTo := THIS^;
IF THIS^.ipStringBuilder = 0 THEN RETURN; END_IF
THIS^.ipStringBuilder.CopySubstringTo(Position, Length, Value);
END_METHOD

(* Copies contents of string builder to given string of any size*)
METHOD CopyTo : I_ReadOnlyStringBuilderAdapter
VAR_INPUT
	Value : ANY;
END_VAR
CopyTo := THIS^;
IF THIS^.ipStringBuilder = 0 THEN RETURN; END_IF
THIS^.ipStringBuilder.CopyTo(Value);
END_METHOD

(* !!!UNSAFE!!! DON'T FORGET TO RELEASE/DELETE FROM	MEMORY WHEN DONE!
 | Get a copy of the internal string buffer at the size of the string length + 1.*)
METHOD GetBuffer : I_ReadOnlyStringBuilderAdapter
VAR_IN_OUT
	pBuffer	: POINTER TO BYTE;
END_VAR
GetBuffer := THIS^;
IF THIS^.ipStringBuilder = 0 THEN RETURN; END_IF
THIS^.ipStringBuilder.GetBuffer(pBuffer);
END_METHOD

(* Retrieves the number of bytes allocated in memory for the string builder's contents.*)
METHOD GetCapacity : I_ReadOnlyStringBuilderAdapter
VAR_OUTPUT
	Capacity	: T_Size;
END_VAR
GetCapacity := THIS^;
Capacity := THIS^.Capacity;
END_METHOD

(* Gets character at specified position in the string builder*)
METHOD GetChar : T_Char
VAR_INPUT
	Position	: T_Size;
END_VAR
IF THIS^.ipStringBuilder = 0 THEN RETURN; END_IF
GetChar := THIS^.ipStringBuilder.GetChar(Position);
END_METHOD

METHOD GetEnumerator : I_Enumerator
VAR_INST
	fbEnumerator : FB_StringBuilderEnumerator(THIS^.ipStringBuilder);
END_VAR
fbEnumerator.FB_init(0,0,THIS^.ipStringBuilder);
GetEnumerator := fbEnumerator;
END_METHOD

(* Retrieves the current size of string builder contents*)
METHOD GetLength : I_ReadOnlyStringBuilderAdapter
VAR_OUTPUT
	Length	: T_Size;
END_VAR
GetLength := THIS^;
Length := THIS^.Length;
END_METHOD

(* Converts contents of string builder to string and returns them*)
METHOD GetString : T_LongString
IF THIS^.ipStringBuilder = 0 THEN RETURN; END_IF
GetString := THIS^.ipStringBuilder.GetString();
END_METHOD

(* Get a subset of characters in the string builder from specified position at specified length and returns them as a string*)
METHOD GetSubstring : T_LongString
VAR_INPUT
	Position	: T_Size;
	Length	: T_Size;
END_VAR
IF THIS^.ipStringBuilder = 0 THEN RETURN; END_IF
GetSubstring := THIS^.ipStringBuilder.GetSubstring(Position, Length);
END_METHOD

(* Current size of string builder contents*)
PROPERTY Length : T_Size
GET
IF THIS^.ipStringBuilder = 0 THEN RETURN; END_IF
Length := THIS^.ipStringBuilder.Length;
END_GET
END_PROPERTY

(* Finds the position of the first instance of a given string in the content's of the string builder from a starting position*)
METHOD Search : I_ReadOnlyStringBuilderAdapter
VAR_INPUT
	sValue	: T_LongString;
	Start_Position	: T_Size;
END_VAR
VAR_OUTPUT
	Position	: T_Size;
END_VAR
Search := THIS^;
IF THIS^.ipStringBuilder = 0 THEN RETURN; END_IF
THIS^.ipStringBuilder.Search(sValue, Start_Position, Position => Position);
END_METHOD

(* Finds the position of the first instance of a given value in the content's of the string builder from a starting position*)
METHOD SearchAny : I_ReadOnlyStringBuilderAdapter
VAR_INPUT
	Value : ANY;
	Start_Position : T_Size;
END_VAR
VAR_OUTPUT
	Position : T_Size := -1;
END_VAR
SearchAny := THIS^;
IF THIS^.ipStringBuilder = 0 THEN RETURN; END_IF
THIS^.ipStringBuilder.SearchAny(Value, Start_Position, Position => Position);
END_METHOD

(* Appends selected characters from the current string builder to the selected string builder*)
METHOD Split : I_ReadOnlyStringBuilderAdapter
VAR_INPUT
	Position, Length : T_Size;
	ipStringBuilder : I_StringBuilder;
END_VAR
Split := THIS^;
IF THIS^.ipStringBuilder = 0 THEN RETURN; END_IF
THIS^.ipStringBuilder.Split(Position, Length, ipStringBuilder);
END_METHOD

END_FUNCTION_BLOCK

// POUs/Examples/P_EnumeratorExample
PROGRAM INTERNAL P_EnumeratorExample
VAR
	bStart				: BOOL;
	sValue				: STRING(255);
	dtTime				: DT :=  DT#2023-5-8-12:55:23;
	fbStringBuilder1,
	fbStringBuilder2	: FB_StringBuilder;
	ipEnumerator		: I_Enumerator;
END_VAR

IF bStart THEN
	bStart := FALSE;
	
	fbStringBuilder1
		.Clear()
		.Append('   I love cats.')
		.Append('The time is: ').AppendAny(dtTime).Append('.')
		.BTrim();
	
	ipEnumerator := fbStringBuilder1.GetEnumerator();
	WHILE ipEnumerator.Next() DO
		fbStringBuilder2.Append(ipEnumerator.Current);
		END_WHILE
		
	sValue := fbStringBuilder2.GetString();
	END_IF

END_PROGRAM

// POUs/Examples/P_StringBuilderExample
PROGRAM INTERNAL P_StringBuilderExample
VAR
	bStart				: BOOL;
	nLn1, nLn2			: T_Size;
	sValue1, sValue2	: STRING(255);
	pString				: POINTER TO STRING;
	fbStringBuilder1,
	fbStringBuilder2	: FB_StringBuilder;
END_VAR

IF bStart THEN
	bStart := FALSE;
	fbStringBuilder2
		.Append(' I hate cats.')
		.GetBuffer(pString);
	
	fbStringBuilder1
		.Clear()
		.Append(' I love cats.')
		.Append(' I love dogs.')
		.AppendBuffer(pString)
		.BTrim()
		.GetLength(Length => nLn1)
		.Replace('cats','dogs',TRUE)
		.Insert(nLn1, ' Anaconda! ')
		.Split(nLn1,100, fbStringBuilder2.Append(' Tigers are cats.'))
		.GetLength(Length => nLn1);
	
	sValue1 := fbStringBuilder1.ToUppercase().GetString();
	sValue2 := fbStringBuilder2
		.ToLowercase()
		.BTrim()
		.GetString();
	
	nLn2 := Tc2_Standard.LEN(sValue1);
	__DELETE(pString);
	END_IF

END_PROGRAM

// POUs/Functions/F_CharToByte
FUNCTION F_CharToByte : BYTE
VAR_INPUT
	Char : T_Char;
END_VAR

F_CharToByte := Char[0];

END_FUNCTION

// POUs/Functions/F_StringBuilder
// String builder function
FUNCTION F_StringBuilder : REFERENCE TO FB_StringBuilder
VAR_STAT
	fbStringBuilder : FB_StringBuilder;
END_VAR

fbStringBuilder.Clear();
F_StringBuilder REF= fbStringBuilder;

END_FUNCTION

// POUs/Functions/F_ToLower
// Converts all alphabetic characters in a string lowercase characters
FUNCTION F_ToLower
VAR_INPUT
	sValue : REFERENCE TO STRING; // String of any size
END_VAR
VAR
	i : T_Size;
END_VAR

WHILE sValue[i] <> 0 DO 
	IF sValue[i] >= 65 AND sValue[i]<= 90 THEN sValue[i] := sValue[i] + 32; END_IF
	i := i + 1;
	END_WHILE

END_FUNCTION

// POUs/Functions/F_TrimWhiteSpace
// Removes all ASCII white space (spaces, tabs, carriage returns, and linefeeds) from the start, end, or both ends of a string
FUNCTION F_TrimWhiteSpace
VAR_INPUT
	sValue : REFERENCE TO STRING; // String of any size
	Location : T_WhitespaceLocation;
END_VAR
VAR
	Start, End, Length, StrLen : T_Size := 0;
	pValue : POINTER TO STRING;
	bMalloced : BOOL := TRUE;
END_VAR

Length := StrLen := F_StrLen(ADR(sValue));

IF Length = 0 THEN RETURN; END_IF
End := Length - 1;

CASE Location OF
	T_WhitespaceLocation.Start:
		
		WHILE ((Start <= End) AND F_IsSpace(F_ByteToChar(sValue[Start]))) DO Start := Start + 1; END_WHILE
	T_WhitespaceLocation.End: 
		WHILE ((End >= Start) AND F_IsSpace(F_ByteToChar(sValue[End]))) DO End := End - 1; END_WHILE
	T_WhitespaceLocation.Both:
		WHILE ((Start <= End) AND F_IsSpace(F_ByteToChar(sValue[Start]))) DO Start := Start  + 1; END_WHILE
		WHILE ((End >= Start) AND F_IsSpace(F_ByteToChar(sValue[End]))) DO End := End - 1; END_WHILE
ELSE
	RETURN;
END_CASE

Length := End - Start + 1;
F_MemMove(ADR(sValue), ADR(sValue[Start]), Length);
sValue[Length] := 0;

END_FUNCTION

// POUs/MAIN
PROGRAM MAIN
VAR
END_VAR

P_EnumeratorExample();
P_AdapterExample();
P_StringBuilderExample();

END_PROGRAM

// Project Information/F_GetCompany
// This function has been automatically generated from the project information.
{attribute 'signature_flag' := '1073741824'}
{attribute 'TcGenerated'}
{attribute 'no-analysis'}
FUNCTION F_GetCompany : WSTRING
VAR_INPUT
	
END_VAR

F_GetCompany := "FisoThemes";

END_FUNCTION

// Project Information/F_GetTitle
// This function has been automatically generated from the project information.
{attribute 'signature_flag' := '1073741824'}
{attribute 'TcGenerated'}
{attribute 'no-analysis'}
FUNCTION F_GetTitle : WSTRING
VAR_INPUT
	
END_VAR

F_GetTitle := "TwinCAT Dynamic String Kit";

END_FUNCTION

// Project Information/F_GetVersion
// This function has been automatically generated from the project information.
{attribute 'signature_flag' := '1073741824'}
{attribute 'TcGenerated'}
{attribute 'no-analysis'}
FUNCTION F_GetVersion : ST_LibVersion
VAR_INPUT
	
END_VAR

F_GetVersion.iMajor := 1;
F_GetVersion.iMinor := 0;
F_GetVersion.iBuild := 1;
F_GetVersion.iRevision := 1;

END_FUNCTION
